   1:  PR[GP1:91,3] = PR[GP1:90,3] + 135.725;
   1:L PR[91] 10mm/sec CNT100;
   1:  PR[GP1:91,1] = PR[GP1:90,1] + 18.371;
   1:  PR[GP1:91,2] = PR[GP1:90,2] + -45.458;
   1:L PR[91] 10mm/sec CNT100;
   1:  PR[GP1:91,1] = PR[GP1:90,1] + 22.302;
   1:  PR[GP1:91,2] = PR[GP1:90,2] + -43.023;
   1:L PR[91] 10mm/sec CNT100;
   1:  PR[GP1:91,1] = PR[GP1:90,1] + 34.257;
   1:  PR[GP1:91,2] = PR[GP1:90,2] + -35.036;
   1:L PR[91] 10mm/sec CNT100;
   1:  PR[GP1:91,1] = PR[GP1:90,1] + 36.457;
   1:  PR[GP1:91,2] = PR[GP1:90,2] + -32.385;
   1:L PR[91] 10mm/sec CNT100;
   1:  PR[GP1:91,1] = PR[GP1:90,1] + 44.453;
   1:  PR[GP1:91,2] = PR[GP1:90,2] + -20.418;
   1:L PR[91] 10mm/sec CNT100;
   1:  PR[GP1:91,1] = PR[GP1:90,1] + 45.837;
   1:  PR[GP1:91,2] = PR[GP1:90,2] + -17.282;
   1:L PR[91] 10mm/sec CNT100;
   1:  PR[GP1:91,1] = PR[GP1:90,1] + 46.320;
   1:  PR[GP1:91,2] = PR[GP1:90,2] + -13.818;
   1:L PR[91] 10mm/sec CNT100;
   1:  PR[GP1:91,1] = PR[GP1:90,1] + 49.129;
   1:  PR[GP1:91,2] = PR[GP1:90,2] + 0.297;
   1:L PR[91] 10mm/sec CNT100;
   1:  PR[GP1:91,1] = PR[GP1:90,1] + 48.653;
   1:  PR[GP1:91,2] = PR[GP1:90,2] + 3.709;
   1:L PR[91] 10mm/sec CNT100;
   1:  PR[GP1:91,1] = PR[GP1:90,1] + 45.844;
   1:  PR[GP1:91,2] = PR[GP1:90,2] + 17.824;
   1:L PR[91] 10mm/sec CNT100;
   1:  PR[GP1:91,1] = PR[GP1:90,1] + 44.453;
   1:  PR[GP1:91,2] = PR[GP1:90,2] + 20.976;
   1:L PR[91] 10mm/sec CNT100;
   1:  PR[GP1:91,1] = PR[GP1:90,1] + 36.457;
   1:  PR[GP1:91,2] = PR[GP1:90,2] + 32.943;
   1:L PR[91] 10mm/sec CNT100;
   1:  PR[GP1:91,1] = PR[GP1:90,1] + 34.257;
   1:  PR[GP1:91,2] = PR[GP1:90,2] + 35.594;
   1:L PR[91] 10mm/sec CNT100;
   1:  PR[GP1:91,1] = PR[GP1:90,1] + 22.302;
   1:  PR[GP1:91,2] = PR[GP1:90,2] + 43.581;
   1:L PR[91] 10mm/sec CNT100;
   1:  PR[GP1:91,1] = PR[GP1:90,1] + 18.371;
   1:  PR[GP1:91,2] = PR[GP1:90,2] + 46.016;
   1:L PR[91] 10mm/sec CNT100;
   1:  PR[GP1:91,1] = PR[GP1:90,1] + 4.284;
   1:  PR[GP1:91,2] = PR[GP1:90,2] + 48.819;
   1:L PR[91] 10mm/sec CNT100;
   1:  PR[GP1:91,1] = PR[GP1:90,1] + -0.264;
   1:  PR[GP1:91,2] = PR[GP1:90,2] + 49.669;
   1:L PR[91] 10mm/sec CNT100;
   1:  PR[GP1:91,1] = PR[GP1:90,1] + -4.810;
   1:  PR[GP1:91,2] = PR[GP1:90,2] + 48.818;
   1:L PR[91] 10mm/sec CNT100;
   1:  PR[GP1:91,1] = PR[GP1:90,1] + -18.898;
   1:  PR[GP1:91,2] = PR[GP1:90,2] + 46.016;
   1:L PR[91] 10mm/sec CNT100;
   1:  PR[GP1:91,1] = PR[GP1:90,1] + -22.828;
   1:  PR[GP1:91,2] = PR[GP1:90,2] + 43.582;
   1:L PR[91] 10mm/sec CNT100;
   1:  PR[GP1:91,1] = PR[GP1:90,1] + -34.783;
   1:  PR[GP1:91,2] = PR[GP1:90,2] + 35.594;
   1:L PR[91] 10mm/sec CNT100;
   1:  PR[GP1:91,1] = PR[GP1:90,1] + -36.984;
   1:  PR[GP1:91,2] = PR[GP1:90,2] + 32.943;
   1:L PR[91] 10mm/sec CNT100;
   1:  PR[GP1:91,1] = PR[GP1:90,1] + -44.979;
   1:  PR[GP1:91,2] = PR[GP1:90,2] + 20.976;
   1:L PR[91] 10mm/sec CNT100;
   1:  PR[GP1:91,1] = PR[GP1:90,1] + -46.364;
   1:  PR[GP1:91,2] = PR[GP1:90,2] + 17.840;
   1:L PR[91] 10mm/sec CNT100;
   1:  PR[GP1:91,1] = PR[GP1:90,1] + -46.847;
   1:  PR[GP1:91,2] = PR[GP1:90,2] + 14.376;
   1:L PR[91] 10mm/sec CNT100;
   1:  PR[GP1:91,1] = PR[GP1:90,1] + -49.655;
   1:  PR[GP1:91,2] = PR[GP1:90,2] + 0.261;
   1:L PR[91] 10mm/sec CNT100;
   1:  PR[GP1:91,1] = PR[GP1:90,1] + -49.179;
   1:  PR[GP1:91,2] = PR[GP1:90,2] + -3.151;
   1:L PR[91] 10mm/sec CNT100;
   1:  PR[GP1:91,1] = PR[GP1:90,1] + -46.371;
   1:  PR[GP1:91,2] = PR[GP1:90,2] + -17.266;
   1:L PR[91] 10mm/sec CNT100;
   1:  PR[GP1:91,1] = PR[GP1:90,1] + -44.979;
   1:  PR[GP1:91,2] = PR[GP1:90,2] + -20.418;
   1:L PR[91] 10mm/sec CNT100;
   1:  PR[GP1:91,1] = PR[GP1:90,1] + -36.984;
   1:  PR[GP1:91,2] = PR[GP1:90,2] + -32.385;
   1:L PR[91] 10mm/sec CNT100;
   1:  PR[GP1:91,1] = PR[GP1:90,1] + -34.783;
   1:  PR[GP1:91,2] = PR[GP1:90,2] + -35.036;
   1:L PR[91] 10mm/sec CNT100;
   1:  PR[GP1:91,1] = PR[GP1:90,1] + -22.828;
   1:  PR[GP1:91,2] = PR[GP1:90,2] + -43.024;
   1:L PR[91] 10mm/sec CNT100;
   1:  PR[GP1:91,1] = PR[GP1:90,1] + -18.901;
   1:  PR[GP1:91,2] = PR[GP1:90,2] + -45.456;
   1:L PR[91] 10mm/sec CNT100;
   1:  PR[GP1:91,1] = PR[GP1:90,1] + -14.348;
   1:  PR[GP1:91,2] = PR[GP1:90,2] + -46.307;
   1:L PR[91] 10mm/sec CNT100;
   1:  PR[GP1:91,1] = PR[GP1:90,1] + -0.261;
   1:  PR[GP1:91,2] = PR[GP1:90,2] + -49.110;
   1:L PR[91] 10mm/sec CNT100;
   1:  PR[GP1:91,1] = PR[GP1:90,1] + 3.182;
   1:  PR[GP1:91,2] = PR[GP1:90,2] + -48.466;
   1:  PR[GP1:91,3] = PR[GP1:90,3] + 136.335;
   1:L PR[91] 10mm/sec CNT100;
   1:  PR[GP1:91,1] = PR[GP1:90,1] + 18.436;
   1:  PR[GP1:91,2] = PR[GP1:90,2] + -45.432;
   1:L PR[91] 10mm/sec CNT100;
   1:  PR[GP1:91,1] = PR[GP1:90,1] + 21.414;
   1:  PR[GP1:91,2] = PR[GP1:90,2] + -43.587;
   1:L PR[91] 10mm/sec CNT100;
   1:  PR[GP1:91,1] = PR[GP1:90,1] + 34.358;
   1:  PR[GP1:91,2] = PR[GP1:90,2] + -34.939;
   1:L PR[91] 10mm/sec CNT100;
   1:  PR[GP1:91,1] = PR[GP1:90,1] + 36.021;
   1:  PR[GP1:91,2] = PR[GP1:90,2] + -32.936;
   1:L PR[91] 10mm/sec CNT100;
   1:  PR[GP1:91,1] = PR[GP1:90,1] + 44.677;
   1:  PR[GP1:91,2] = PR[GP1:90,2] + -19.980;
   1:L PR[91] 10mm/sec CNT100;
   1:  PR[GP1:91,1] = PR[GP1:90,1] + 45.721;
   1:  PR[GP1:91,2] = PR[GP1:90,2] + -17.615;
   1:L PR[91] 10mm/sec CNT100;
   1:  PR[GP1:91,1] = PR[GP1:90,1] + 46.088;
   1:  PR[GP1:91,2] = PR[GP1:90,2] + -14.985;
   1:L PR[91] 10mm/sec CNT100;
   1:  PR[GP1:91,1] = PR[GP1:90,1] + 49.129;
   1:  PR[GP1:91,2] = PR[GP1:90,2] + 0.297;
   1:L PR[91] 10mm/sec CNT100;
   1:  PR[GP1:91,1] = PR[GP1:90,1] + 48.769;
   1:  PR[GP1:91,2] = PR[GP1:90,2] + 2.874;
   1:L PR[91] 10mm/sec CNT100;
   1:  PR[GP1:91,1] = PR[GP1:90,1] + 45.729;
   1:  PR[GP1:91,2] = PR[GP1:90,2] + 18.157;
   1:L PR[91] 10mm/sec CNT100;
   1:  PR[GP1:91,1] = PR[GP1:90,1] + 44.677;
   1:  PR[GP1:91,2] = PR[GP1:90,2] + 20.538;
   1:L PR[91] 10mm/sec CNT100;
   1:  PR[GP1:91,1] = PR[GP1:90,1] + 36.021;
   1:  PR[GP1:91,2] = PR[GP1:90,2] + 33.494;
   1:L PR[91] 10mm/sec CNT100;
   1:  PR[GP1:91,1] = PR[GP1:90,1] + 34.358;
   1:  PR[GP1:91,2] = PR[GP1:90,2] + 35.497;
   1:L PR[91] 10mm/sec CNT100;
   1:  PR[GP1:91,1] = PR[GP1:90,1] + 21.414;
   1:  PR[GP1:91,2] = PR[GP1:90,2] + 44.145;
   1:L PR[91] 10mm/sec CNT100;
   1:  PR[GP1:91,1] = PR[GP1:90,1] + 18.436;
   1:  PR[GP1:91,2] = PR[GP1:90,2] + 45.990;
   1:L PR[91] 10mm/sec CNT100;
   1:  PR[GP1:91,1] = PR[GP1:90,1] + 3.182;
   1:  PR[GP1:91,2] = PR[GP1:90,2] + 49.025;
   1:L PR[91] 10mm/sec CNT100;
   1:  PR[GP1:91,1] = PR[GP1:90,1] + -0.264;
   1:  PR[GP1:91,2] = PR[GP1:90,2] + 49.669;
   1:L PR[91] 10mm/sec CNT100;
   1:  PR[GP1:91,1] = PR[GP1:90,1] + -3.708;
   1:  PR[GP1:91,2] = PR[GP1:90,2] + 49.024;
   1:L PR[91] 10mm/sec CNT100;
   1:  PR[GP1:91,1] = PR[GP1:90,1] + -18.963;
   1:  PR[GP1:91,2] = PR[GP1:90,2] + 45.989;
   1:L PR[91] 10mm/sec CNT100;
   1:  PR[GP1:91,1] = PR[GP1:90,1] + -21.940;
   1:  PR[GP1:91,2] = PR[GP1:90,2] + 44.146;
   1:L PR[91] 10mm/sec CNT100;
   1:  PR[GP1:91,1] = PR[GP1:90,1] + -34.885;
   1:  PR[GP1:91,2] = PR[GP1:90,2] + 35.497;
   1:L PR[91] 10mm/sec CNT100;
   1:  PR[GP1:91,1] = PR[GP1:90,1] + -36.547;
   1:  PR[GP1:91,2] = PR[GP1:90,2] + 33.495;
   1:L PR[91] 10mm/sec CNT100;
   1:  PR[GP1:91,1] = PR[GP1:90,1] + -45.204;
   1:  PR[GP1:91,2] = PR[GP1:90,2] + 20.538;
   1:L PR[91] 10mm/sec CNT100;
   1:  PR[GP1:91,1] = PR[GP1:90,1] + -46.248;
   1:  PR[GP1:91,2] = PR[GP1:90,2] + 18.173;
   1:L PR[91] 10mm/sec CNT100;
   1:  PR[GP1:91,1] = PR[GP1:90,1] + -46.615;
   1:  PR[GP1:91,2] = PR[GP1:90,2] + 15.543;
   1:L PR[91] 10mm/sec CNT100;
   1:  PR[GP1:91,1] = PR[GP1:90,1] + -49.655;
   1:  PR[GP1:91,2] = PR[GP1:90,2] + 0.261;
   1:L PR[91] 10mm/sec CNT100;
   1:  PR[GP1:91,1] = PR[GP1:90,1] + -49.295;
   1:  PR[GP1:91,2] = PR[GP1:90,2] + -2.316;
   1:L PR[91] 10mm/sec CNT100;
   1:  PR[GP1:91,1] = PR[GP1:90,1] + -46.255;
   1:  PR[GP1:91,2] = PR[GP1:90,2] + -17.599;
   1:L PR[91] 10mm/sec CNT100;
   1:  PR[GP1:91,1] = PR[GP1:90,1] + -45.204;
   1:  PR[GP1:91,2] = PR[GP1:90,2] + -19.980;
   1:L PR[91] 10mm/sec CNT100;
   1:  PR[GP1:91,1] = PR[GP1:90,1] + -36.547;
   1:  PR[GP1:91,2] = PR[GP1:90,2] + -32.937;
   1:L PR[91] 10mm/sec CNT100;
   1:  PR[GP1:91,1] = PR[GP1:90,1] + -34.885;
   1:  PR[GP1:91,2] = PR[GP1:90,2] + -34.939;
   1:L PR[91] 10mm/sec CNT100;
   1:  PR[GP1:91,1] = PR[GP1:90,1] + -21.940;
   1:  PR[GP1:91,2] = PR[GP1:90,2] + -43.588;
   1:L PR[91] 10mm/sec CNT100;
   1:  PR[GP1:91,1] = PR[GP1:90,1] + -18.966;
   1:  PR[GP1:91,2] = PR[GP1:90,2] + -45.429;
   1:L PR[91] 10mm/sec CNT100;
   1:  PR[GP1:91,1] = PR[GP1:90,1] + -15.515;
   1:  PR[GP1:91,2] = PR[GP1:90,2] + -46.075;
   1:L PR[91] 10mm/sec CNT100;
   1:  PR[GP1:91,1] = PR[GP1:90,1] + -0.260;
   1:  PR[GP1:91,2] = PR[GP1:90,2] + -49.110;
   1:L PR[91] 10mm/sec CNT100;
   1:  PR[GP1:91,1] = PR[GP1:90,1] + 2.080;
   1:  PR[GP1:91,2] = PR[GP1:90,2] + -48.672;
   1:  PR[GP1:91,3] = PR[GP1:90,3] + 136.945;
   1:L PR[91] 10mm/sec CNT100;
   1:  PR[GP1:91,1] = PR[GP1:90,1] + 18.502;
   1:  PR[GP1:91,2] = PR[GP1:90,2] + -45.405;
   1:L PR[91] 10mm/sec CNT100;
   1:  PR[GP1:91,1] = PR[GP1:90,1] + 20.526;
   1:  PR[GP1:91,2] = PR[GP1:90,2] + -44.152;
   1:L PR[91] 10mm/sec CNT100;
   1:  PR[GP1:91,1] = PR[GP1:90,1] + 34.460;
   1:  PR[GP1:91,2] = PR[GP1:90,2] + -34.842;
   1:L PR[91] 10mm/sec CNT100;
   1:  PR[GP1:91,1] = PR[GP1:90,1] + 35.584;
   1:  PR[GP1:91,2] = PR[GP1:90,2] + -33.488;
   1:L PR[91] 10mm/sec CNT100;
   1:  PR[GP1:91,1] = PR[GP1:90,1] + 44.902;
   1:  PR[GP1:91,2] = PR[GP1:90,2] + -19.542;
   1:L PR[91] 10mm/sec CNT100;
   1:  PR[GP1:91,1] = PR[GP1:90,1] + 45.606;
   1:  PR[GP1:91,2] = PR[GP1:90,2] + -17.948;
   1:L PR[91] 10mm/sec CNT100;
   1:  PR[GP1:91,1] = PR[GP1:90,1] + 45.856;
   1:  PR[GP1:91,2] = PR[GP1:90,2] + -16.152;
   1:L PR[91] 10mm/sec CNT100;
   1:  PR[GP1:91,1] = PR[GP1:90,1] + 49.129;
   1:  PR[GP1:91,2] = PR[GP1:90,2] + 0.297;
   1:L PR[91] 10mm/sec CNT100;
   1:  PR[GP1:91,1] = PR[GP1:90,1] + 48.885;
   1:  PR[GP1:91,2] = PR[GP1:90,2] + 2.040;
   1:L PR[91] 10mm/sec CNT100;
   1:  PR[GP1:91,1] = PR[GP1:90,1] + 45.613;
   1:  PR[GP1:91,2] = PR[GP1:90,2] + 18.489;
   1:L PR[91] 10mm/sec CNT100;
   1:  PR[GP1:91,1] = PR[GP1:90,1] + 44.902;
   1:  PR[GP1:91,2] = PR[GP1:90,2] + 20.100;
   1:L PR[91] 10mm/sec CNT100;
   1:  PR[GP1:91,1] = PR[GP1:90,1] + 35.584;
   1:  PR[GP1:91,2] = PR[GP1:90,2] + 34.046;
   1:L PR[91] 10mm/sec CNT100;
   1:  PR[GP1:91,1] = PR[GP1:90,1] + 34.460;
   1:  PR[GP1:91,2] = PR[GP1:90,2] + 35.400;
   1:L PR[91] 10mm/sec CNT100;
   1:  PR[GP1:91,1] = PR[GP1:90,1] + 20.526;
   1:  PR[GP1:91,2] = PR[GP1:90,2] + 44.710;
   1:L PR[91] 10mm/sec CNT100;
   1:  PR[GP1:91,1] = PR[GP1:90,1] + 18.502;
   1:  PR[GP1:91,2] = PR[GP1:90,2] + 45.963;
   1:L PR[91] 10mm/sec CNT100;
   1:  PR[GP1:91,1] = PR[GP1:90,1] + 2.080;
   1:  PR[GP1:91,2] = PR[GP1:90,2] + 49.230;
   1:L PR[91] 10mm/sec CNT100;
   1:  PR[GP1:91,1] = PR[GP1:90,1] + -0.264;
   1:  PR[GP1:91,2] = PR[GP1:90,2] + 49.669;
   1:L PR[91] 10mm/sec CNT100;
   1:  PR[GP1:91,1] = PR[GP1:90,1] + -2.606;
   1:  PR[GP1:91,2] = PR[GP1:90,2] + 49.230;
   1:L PR[91] 10mm/sec CNT100;
   1:  PR[GP1:91,1] = PR[GP1:90,1] + -19.028;
   1:  PR[GP1:91,2] = PR[GP1:90,2] + 45.963;
   1:L PR[91] 10mm/sec CNT100;
   1:  PR[GP1:91,1] = PR[GP1:90,1] + -21.052;
   1:  PR[GP1:91,2] = PR[GP1:90,2] + 44.710;
   1:L PR[91] 10mm/sec CNT100;
   1:  PR[GP1:91,1] = PR[GP1:90,1] + -34.986;
   1:  PR[GP1:91,2] = PR[GP1:90,2] + 35.400;
   1:L PR[91] 10mm/sec CNT100;
   1:  PR[GP1:91,1] = PR[GP1:90,1] + -36.110;
   1:  PR[GP1:91,2] = PR[GP1:90,2] + 34.046;
   1:L PR[91] 10mm/sec CNT100;
   1:  PR[GP1:91,1] = PR[GP1:90,1] + -45.428;
   1:  PR[GP1:91,2] = PR[GP1:90,2] + 20.100;
   1:L PR[91] 10mm/sec CNT100;
   1:  PR[GP1:91,1] = PR[GP1:90,1] + -46.132;
   1:  PR[GP1:91,2] = PR[GP1:90,2] + 18.506;
   1:L PR[91] 10mm/sec CNT100;
   1:  PR[GP1:91,1] = PR[GP1:90,1] + -46.382;
   1:  PR[GP1:91,2] = PR[GP1:90,2] + 16.711;
   1:L PR[91] 10mm/sec CNT100;
   1:  PR[GP1:91,1] = PR[GP1:90,1] + -49.655;
   1:  PR[GP1:91,2] = PR[GP1:90,2] + 0.261;
   1:L PR[91] 10mm/sec CNT100;
   1:  PR[GP1:91,1] = PR[GP1:90,1] + -49.412;
   1:  PR[GP1:91,2] = PR[GP1:90,2] + -1.482;
   1:L PR[91] 10mm/sec CNT100;
   1:  PR[GP1:91,1] = PR[GP1:90,1] + -46.139;
   1:  PR[GP1:91,2] = PR[GP1:90,2] + -17.931;
   1:L PR[91] 10mm/sec CNT100;
   1:  PR[GP1:91,1] = PR[GP1:90,1] + -45.428;
   1:  PR[GP1:91,2] = PR[GP1:90,2] + -19.542;
   1:L PR[91] 10mm/sec CNT100;
   1:  PR[GP1:91,1] = PR[GP1:90,1] + -36.110;
   1:  PR[GP1:91,2] = PR[GP1:90,2] + -33.488;
   1:L PR[91] 10mm/sec CNT100;
   1:  PR[GP1:91,1] = PR[GP1:90,1] + -34.986;
   1:  PR[GP1:91,2] = PR[GP1:90,2] + -34.842;
   1:L PR[91] 10mm/sec CNT100;
   1:  PR[GP1:91,1] = PR[GP1:90,1] + -21.052;
   1:  PR[GP1:91,2] = PR[GP1:90,2] + -44.152;
   1:L PR[91] 10mm/sec CNT100;
   1:  PR[GP1:91,1] = PR[GP1:90,1] + -19.031;
   1:  PR[GP1:91,2] = PR[GP1:90,2] + -45.403;
   1:L PR[91] 10mm/sec CNT100;
   1:  PR[GP1:91,1] = PR[GP1:90,1] + -16.682;
   1:  PR[GP1:91,2] = PR[GP1:90,2] + -45.843;
   1:L PR[91] 10mm/sec CNT100;
   1:  PR[GP1:91,1] = PR[GP1:90,1] + -0.260;
   1:  PR[GP1:91,2] = PR[GP1:90,2] + -49.110;
   1:L PR[91] 10mm/sec CNT100;
   1:  PR[GP1:91,1] = PR[GP1:90,1] + 0.978;
   1:  PR[GP1:91,2] = PR[GP1:90,2] + -48.878;
   1:  PR[GP1:91,3] = PR[GP1:90,3] + 137.555;
   1:L PR[91] 10mm/sec CNT100;
   1:  PR[GP1:91,1] = PR[GP1:90,1] + 18.567;
   1:  PR[GP1:91,2] = PR[GP1:90,2] + -45.379;
   1:L PR[91] 10mm/sec CNT100;
   1:  PR[GP1:91,1] = PR[GP1:90,1] + 19.638;
   1:  PR[GP1:91,2] = PR[GP1:90,2] + -44.716;
   1:L PR[91] 10mm/sec CNT100;
   1:  PR[GP1:91,1] = PR[GP1:90,1] + 34.561;
   1:  PR[GP1:91,2] = PR[GP1:90,2] + -34.745;
   1:L PR[91] 10mm/sec CNT100;
   1:  PR[GP1:91,1] = PR[GP1:90,1] + 35.147;
   1:  PR[GP1:91,2] = PR[GP1:90,2] + -34.039;
   1:L PR[91] 10mm/sec CNT100;
   1:  PR[GP1:91,1] = PR[GP1:90,1] + 45.126;
   1:  PR[GP1:91,2] = PR[GP1:90,2] + -19.104;
   1:L PR[91] 10mm/sec CNT100;
   1:  PR[GP1:91,1] = PR[GP1:90,1] + 45.490;
   1:  PR[GP1:91,2] = PR[GP1:90,2] + -18.280;
   1:L PR[91] 10mm/sec CNT100;
   1:  PR[GP1:91,1] = PR[GP1:90,1] + 45.624;
   1:  PR[GP1:91,2] = PR[GP1:90,2] + -17.320;
   1:L PR[91] 10mm/sec CNT100;
   1:  PR[GP1:91,1] = PR[GP1:90,1] + 49.129;
   1:  PR[GP1:91,2] = PR[GP1:90,2] + 0.297;
   1:L PR[91] 10mm/sec CNT100;
   1:  PR[GP1:91,1] = PR[GP1:90,1] + 49.002;
   1:  PR[GP1:91,2] = PR[GP1:90,2] + 1.205;
   1:L PR[91] 10mm/sec CNT100;
   1:  PR[GP1:91,1] = PR[GP1:90,1] + 45.497;
   1:  PR[GP1:91,2] = PR[GP1:90,2] + 18.822;
   1:L PR[91] 10mm/sec CNT100;
   1:  PR[GP1:91,1] = PR[GP1:90,1] + 45.126;
   1:  PR[GP1:91,2] = PR[GP1:90,2] + 19.662;
   1:L PR[91] 10mm/sec CNT100;
   1:  PR[GP1:91,1] = PR[GP1:90,1] + 35.147;
   1:  PR[GP1:91,2] = PR[GP1:90,2] + 34.597;
   1:L PR[91] 10mm/sec CNT100;
   1:  PR[GP1:91,1] = PR[GP1:90,1] + 34.561;
   1:  PR[GP1:91,2] = PR[GP1:90,2] + 35.303;
   1:L PR[91] 10mm/sec CNT100;
   1:  PR[GP1:91,1] = PR[GP1:90,1] + 19.638;
   1:  PR[GP1:91,2] = PR[GP1:90,2] + 45.274;
   1:L PR[91] 10mm/sec CNT100;
   1:  PR[GP1:91,1] = PR[GP1:90,1] + 18.567;
   1:  PR[GP1:91,2] = PR[GP1:90,2] + 45.937;
   1:L PR[91] 10mm/sec CNT100;
   1:  PR[GP1:91,1] = PR[GP1:90,1] + 0.978;
   1:  PR[GP1:91,2] = PR[GP1:90,2] + 49.437;
   1:L PR[91] 10mm/sec CNT100;
   1:  PR[GP1:91,1] = PR[GP1:90,1] + -0.263;
   1:  PR[GP1:91,2] = PR[GP1:90,2] + 49.669;
   1:L PR[91] 10mm/sec CNT100;
   1:  PR[GP1:91,1] = PR[GP1:90,1] + -1.504;
   1:  PR[GP1:91,2] = PR[GP1:90,2] + 49.437;
   1:L PR[91] 10mm/sec CNT100;
   1:  PR[GP1:91,1] = PR[GP1:90,1] + -19.093;
   1:  PR[GP1:91,2] = PR[GP1:90,2] + 45.937;
   1:L PR[91] 10mm/sec CNT100;
   1:  PR[GP1:91,1] = PR[GP1:90,1] + -20.164;
   1:  PR[GP1:91,2] = PR[GP1:90,2] + 45.274;
   1:L PR[91] 10mm/sec CNT100;
   1:  PR[GP1:91,1] = PR[GP1:90,1] + -35.088;
   1:  PR[GP1:91,2] = PR[GP1:90,2] + 35.303;
   1:L PR[91] 10mm/sec CNT100;
   1:  PR[GP1:91,1] = PR[GP1:90,1] + -35.674;
   1:  PR[GP1:91,2] = PR[GP1:90,2] + 34.597;
   1:L PR[91] 10mm/sec CNT100;
   1:  PR[GP1:91,1] = PR[GP1:90,1] + -45.653;
   1:  PR[GP1:91,2] = PR[GP1:90,2] + 19.662;
   1:L PR[91] 10mm/sec CNT100;
   1:  PR[GP1:91,1] = PR[GP1:90,1] + -46.016;
   1:  PR[GP1:91,2] = PR[GP1:90,2] + 18.838;
   1:L PR[91] 10mm/sec CNT100;
   1:  PR[GP1:91,1] = PR[GP1:90,1] + -46.150;
   1:  PR[GP1:91,2] = PR[GP1:90,2] + 17.878;
   1:L PR[91] 10mm/sec CNT100;
   1:  PR[GP1:91,1] = PR[GP1:90,1] + -49.655;
   1:  PR[GP1:91,2] = PR[GP1:90,2] + 0.261;
   1:L PR[91] 10mm/sec CNT100;
   1:  PR[GP1:91,1] = PR[GP1:90,1] + -49.528;
   1:  PR[GP1:91,2] = PR[GP1:90,2] + -0.647;
   1:L PR[91] 10mm/sec CNT100;
   1:  PR[GP1:91,1] = PR[GP1:90,1] + -46.023;
   1:  PR[GP1:91,2] = PR[GP1:90,2] + -18.264;
   1:L PR[91] 10mm/sec CNT100;
   1:  PR[GP1:91,1] = PR[GP1:90,1] + -45.653;
   1:  PR[GP1:91,2] = PR[GP1:90,2] + -19.104;
   1:L PR[91] 10mm/sec CNT100;
   1:  PR[GP1:91,1] = PR[GP1:90,1] + -35.674;
   1:  PR[GP1:91,2] = PR[GP1:90,2] + -34.039;
   1:L PR[91] 10mm/sec CNT100;
   1:  PR[GP1:91,1] = PR[GP1:90,1] + -35.088;
   1:  PR[GP1:91,2] = PR[GP1:90,2] + -34.745;
   1:L PR[91] 10mm/sec CNT100;
   1:  PR[GP1:91,1] = PR[GP1:90,1] + -20.164;
   1:  PR[GP1:91,2] = PR[GP1:90,2] + -44.716;
   1:L PR[91] 10mm/sec CNT100;
   1:  PR[GP1:91,1] = PR[GP1:90,1] + -19.096;
   1:  PR[GP1:91,2] = PR[GP1:90,2] + -45.377;
   1:L PR[91] 10mm/sec CNT100;
   1:  PR[GP1:91,1] = PR[GP1:90,1] + -17.849;
   1:  PR[GP1:91,2] = PR[GP1:90,2] + -45.611;
   1:L PR[91] 10mm/sec CNT100;
   1:  PR[GP1:91,1] = PR[GP1:90,1] + -0.260;
   1:  PR[GP1:91,2] = PR[GP1:90,2] + -49.110;
   1:L PR[91] 10mm/sec CNT100;
   1:  PR[GP1:91,1] = PR[GP1:90,1] + 18.622;
   1:  PR[GP1:91,2] = PR[GP1:90,2] + -45.355;
   1:  PR[GP1:91,3] = PR[GP1:90,3] + 138.165;
   1:L PR[91] 10mm/sec CNT100;
   1:  PR[GP1:91,1] = PR[GP1:90,1] + 34.663;
   1:  PR[GP1:91,2] = PR[GP1:90,2] + -34.648;
   1:L PR[91] 10mm/sec CNT100;
   1:  PR[GP1:91,1] = PR[GP1:90,1] + 34.711;
   1:  PR[GP1:91,2] = PR[GP1:90,2] + -34.590;
   1:L PR[91] 10mm/sec CNT100;
   1:  PR[GP1:91,1] = PR[GP1:90,1] + 45.351;
   1:  PR[GP1:91,2] = PR[GP1:90,2] + -18.665;
   1:L PR[91] 10mm/sec CNT100;
   1:  PR[GP1:91,1] = PR[GP1:90,1] + 45.374;
   1:  PR[GP1:91,2] = PR[GP1:90,2] + -18.613;
   1:L PR[91] 10mm/sec CNT100;
   1:  PR[GP1:91,1] = PR[GP1:90,1] + 45.392;
   1:  PR[GP1:91,2] = PR[GP1:90,2] + -18.487;
   1:L PR[91] 10mm/sec CNT100;
   1:  PR[GP1:91,1] = PR[GP1:90,1] + 49.129;
   1:  PR[GP1:91,2] = PR[GP1:90,2] + 0.297;
   1:L PR[91] 10mm/sec CNT100;
   1:  PR[GP1:91,1] = PR[GP1:90,1] + 49.118;
   1:  PR[GP1:91,2] = PR[GP1:90,2] + 0.371;
   1:L PR[91] 10mm/sec CNT100;
   1:  PR[GP1:91,1] = PR[GP1:90,1] + 45.381;
   1:  PR[GP1:91,2] = PR[GP1:90,2] + 19.155;
   1:L PR[91] 10mm/sec CNT100;
   1:  PR[GP1:91,1] = PR[GP1:90,1] + 45.351;
   1:  PR[GP1:91,2] = PR[GP1:90,2] + 19.224;
   1:L PR[91] 10mm/sec CNT100;
   1:  PR[GP1:91,1] = PR[GP1:90,1] + 34.711;
   1:  PR[GP1:91,2] = PR[GP1:90,2] + 35.149;
   1:L PR[91] 10mm/sec CNT100;
   1:  PR[GP1:91,1] = PR[GP1:90,1] + 34.663;
   1:  PR[GP1:91,2] = PR[GP1:90,2] + 35.206;
   1:L PR[91] 10mm/sec CNT100;
   1:  PR[GP1:91,1] = PR[GP1:90,1] + 18.622;
   1:  PR[GP1:91,2] = PR[GP1:90,2] + 45.913;
   1:L PR[91] 10mm/sec CNT100;
   1:  PR[GP1:91,1] = PR[GP1:90,1] + -0.263;
   1:  PR[GP1:91,2] = PR[GP1:90,2] + 49.667;
   1:L PR[91] 10mm/sec CNT100;
   1:  PR[GP1:91,1] = PR[GP1:90,1] + -19.148;
   1:  PR[GP1:91,2] = PR[GP1:90,2] + 45.913;
   1:L PR[91] 10mm/sec CNT100;
   1:  PR[GP1:91,1] = PR[GP1:90,1] + -35.189;
   1:  PR[GP1:91,2] = PR[GP1:90,2] + 35.206;
   1:L PR[91] 10mm/sec CNT100;
   1:  PR[GP1:91,1] = PR[GP1:90,1] + -35.237;
   1:  PR[GP1:91,2] = PR[GP1:90,2] + 35.149;
   1:L PR[91] 10mm/sec CNT100;
   1:  PR[GP1:91,1] = PR[GP1:90,1] + -45.877;
   1:  PR[GP1:91,2] = PR[GP1:90,2] + 19.224;
   1:L PR[91] 10mm/sec CNT100;
   1:  PR[GP1:91,1] = PR[GP1:90,1] + -45.900;
   1:  PR[GP1:91,2] = PR[GP1:90,2] + 19.171;
   1:L PR[91] 10mm/sec CNT100;
   1:  PR[GP1:91,1] = PR[GP1:90,1] + -45.918;
   1:  PR[GP1:91,2] = PR[GP1:90,2] + 19.045;
   1:L PR[91] 10mm/sec CNT100;
   1:  PR[GP1:91,1] = PR[GP1:90,1] + -49.655;
   1:  PR[GP1:91,2] = PR[GP1:90,2] + 0.261;
   1:L PR[91] 10mm/sec CNT100;
   1:  PR[GP1:91,1] = PR[GP1:90,1] + -49.645;
   1:  PR[GP1:91,2] = PR[GP1:90,2] + 0.188;
   1:L PR[91] 10mm/sec CNT100;
   1:  PR[GP1:91,1] = PR[GP1:90,1] + -45.907;
   1:  PR[GP1:91,2] = PR[GP1:90,2] + -18.597;
   1:L PR[91] 10mm/sec CNT100;
   1:  PR[GP1:91,1] = PR[GP1:90,1] + -45.877;
   1:  PR[GP1:91,2] = PR[GP1:90,2] + -18.665;
   1:L PR[91] 10mm/sec CNT100;
   1:  PR[GP1:91,1] = PR[GP1:90,1] + -35.237;
   1:  PR[GP1:91,2] = PR[GP1:90,2] + -34.590;
   1:L PR[91] 10mm/sec CNT100;
   1:  PR[GP1:91,1] = PR[GP1:90,1] + -35.189;
   1:  PR[GP1:91,2] = PR[GP1:90,2] + -34.648;
   1:L PR[91] 10mm/sec CNT100;
   1:  PR[GP1:91,1] = PR[GP1:90,1] + -19.148;
   1:  PR[GP1:91,2] = PR[GP1:90,2] + -45.355;
   1:L PR[91] 10mm/sec CNT100;
   1:  PR[GP1:91,1] = PR[GP1:90,1] + -0.263;
   1:  PR[GP1:91,2] = PR[GP1:90,2] + -49.109;
   1:L PR[91] 10mm/sec CNT100;
   1:  PR[GP1:91,1] = PR[GP1:90,1] + 18.622;
   1:  PR[GP1:91,2] = PR[GP1:90,2] + -45.355;
   1:L PR[91] 10mm/sec CNT100;
   1:  PR[GP1:91,1] = PR[GP1:90,1] + 34.663;
   1:  PR[GP1:91,2] = PR[GP1:90,2] + -34.648;
   1:L PR[91] 10mm/sec CNT100;
   1:  PR[GP1:91,1] = PR[GP1:90,1] + 34.711;
   1:  PR[GP1:91,2] = PR[GP1:90,2] + -34.590;
   1:L PR[91] 10mm/sec CNT100;
   1:  PR[GP1:91,1] = PR[GP1:90,1] + 45.351;
   1:  PR[GP1:91,2] = PR[GP1:90,2] + -18.665;
   1:L PR[91] 10mm/sec CNT100;
   1:  PR[GP1:91,1] = PR[GP1:90,1] + 45.374;
   1:  PR[GP1:91,2] = PR[GP1:90,2] + -18.613;
   1:L PR[91] 10mm/sec CNT100;
   1:  PR[GP1:91,1] = PR[GP1:90,1] + 45.392;
   1:  PR[GP1:91,2] = PR[GP1:90,2] + -18.487;
   1:L PR[91] 10mm/sec CNT100;
   1:  PR[GP1:91,1] = PR[GP1:90,1] + 49.129;
   1:  PR[GP1:91,2] = PR[GP1:90,2] + 0.297;
   1:L PR[91] 10mm/sec CNT100;
   1:  PR[GP1:91,1] = PR[GP1:90,1] + 49.118;
   1:  PR[GP1:91,2] = PR[GP1:90,2] + 0.371;
   1:L PR[91] 10mm/sec CNT100;
   1:  PR[GP1:91,1] = PR[GP1:90,1] + 45.381;
   1:  PR[GP1:91,2] = PR[GP1:90,2] + 19.155;
   1:L PR[91] 10mm/sec CNT100;
   1:  PR[GP1:91,1] = PR[GP1:90,1] + 45.351;
   1:  PR[GP1:91,2] = PR[GP1:90,2] + 19.224;
   1:L PR[91] 10mm/sec CNT100;
   1:  PR[GP1:91,1] = PR[GP1:90,1] + 34.711;
   1:  PR[GP1:91,2] = PR[GP1:90,2] + 35.149;
   1:L PR[91] 10mm/sec CNT100;
   1:  PR[GP1:91,1] = PR[GP1:90,1] + 34.663;
   1:  PR[GP1:91,2] = PR[GP1:90,2] + 35.206;
   1:L PR[91] 10mm/sec CNT100;
   1:  PR[GP1:91,1] = PR[GP1:90,1] + 18.622;
   1:  PR[GP1:91,2] = PR[GP1:90,2] + 45.913;
   1:L PR[91] 10mm/sec CNT100;
   1:  PR[GP1:91,1] = PR[GP1:90,1] + -0.263;
   1:  PR[GP1:91,2] = PR[GP1:90,2] + 49.667;
   1:L PR[91] 10mm/sec CNT100;
   1:  PR[GP1:91,1] = PR[GP1:90,1] + -19.148;
   1:  PR[GP1:91,2] = PR[GP1:90,2] + 45.913;
   1:L PR[91] 10mm/sec CNT100;
   1:  PR[GP1:91,1] = PR[GP1:90,1] + -35.189;
   1:  PR[GP1:91,2] = PR[GP1:90,2] + 35.206;
   1:L PR[91] 10mm/sec CNT100;
   1:  PR[GP1:91,1] = PR[GP1:90,1] + -35.237;
   1:  PR[GP1:91,2] = PR[GP1:90,2] + 35.149;
   1:L PR[91] 10mm/sec CNT100;
   1:  PR[GP1:91,1] = PR[GP1:90,1] + -45.877;
   1:  PR[GP1:91,2] = PR[GP1:90,2] + 19.224;
   1:L PR[91] 10mm/sec CNT100;
   1:  PR[GP1:91,1] = PR[GP1:90,1] + -45.900;
   1:  PR[GP1:91,2] = PR[GP1:90,2] + 19.171;
   1:L PR[91] 10mm/sec CNT100;
   1:  PR[GP1:91,1] = PR[GP1:90,1] + -45.918;
   1:  PR[GP1:91,2] = PR[GP1:90,2] + 19.045;
   1:L PR[91] 10mm/sec CNT100;
   1:  PR[GP1:91,1] = PR[GP1:90,1] + -49.655;
   1:  PR[GP1:91,2] = PR[GP1:90,2] + 0.261;
   1:L PR[91] 10mm/sec CNT100;
   1:  PR[GP1:91,1] = PR[GP1:90,1] + -49.645;
   1:  PR[GP1:91,2] = PR[GP1:90,2] + 0.188;
   1:L PR[91] 10mm/sec CNT100;
   1:  PR[GP1:91,1] = PR[GP1:90,1] + -45.907;
   1:  PR[GP1:91,2] = PR[GP1:90,2] + -18.597;
   1:L PR[91] 10mm/sec CNT100;
   1:  PR[GP1:91,1] = PR[GP1:90,1] + -45.877;
   1:  PR[GP1:91,2] = PR[GP1:90,2] + -18.665;
   1:L PR[91] 10mm/sec CNT100;
   1:  PR[GP1:91,1] = PR[GP1:90,1] + -35.237;
   1:  PR[GP1:91,2] = PR[GP1:90,2] + -34.590;
   1:L PR[91] 10mm/sec CNT100;
   1:  PR[GP1:91,1] = PR[GP1:90,1] + -35.189;
   1:  PR[GP1:91,2] = PR[GP1:90,2] + -34.648;
   1:L PR[91] 10mm/sec CNT100;
   1:  PR[GP1:91,1] = PR[GP1:90,1] + -19.148;
   1:  PR[GP1:91,2] = PR[GP1:90,2] + -45.355;
   1:L PR[91] 10mm/sec CNT100;
   1:  PR[GP1:91,1] = PR[GP1:90,1] + -0.263;
   1:  PR[GP1:91,2] = PR[GP1:90,2] + -49.109;
   1:L PR[91] 10mm/sec CNT100;
   1:  CALL HOME_ALL;
/POS
/END
